SYSTEM FLASH_Lecture (* Remote Flasher Test System Configuration *)
  (* Standard: 61499-1 *)
  (* Version 0.1, 2009-03-05, JHC, Holobloc Inc., Deleted Application. *)
  (* Version 0.0, 2004-01-10, JHC, Rockwell Automation, Modified from FLASHERT_TESTD. *)
  DEVICE CTL_PANEL : FRAME_DEVICE(BOUNDS := [50,100,325,100], GRID := [1,1])
    RESOURCE RES1 : PANEL_RESOURCE
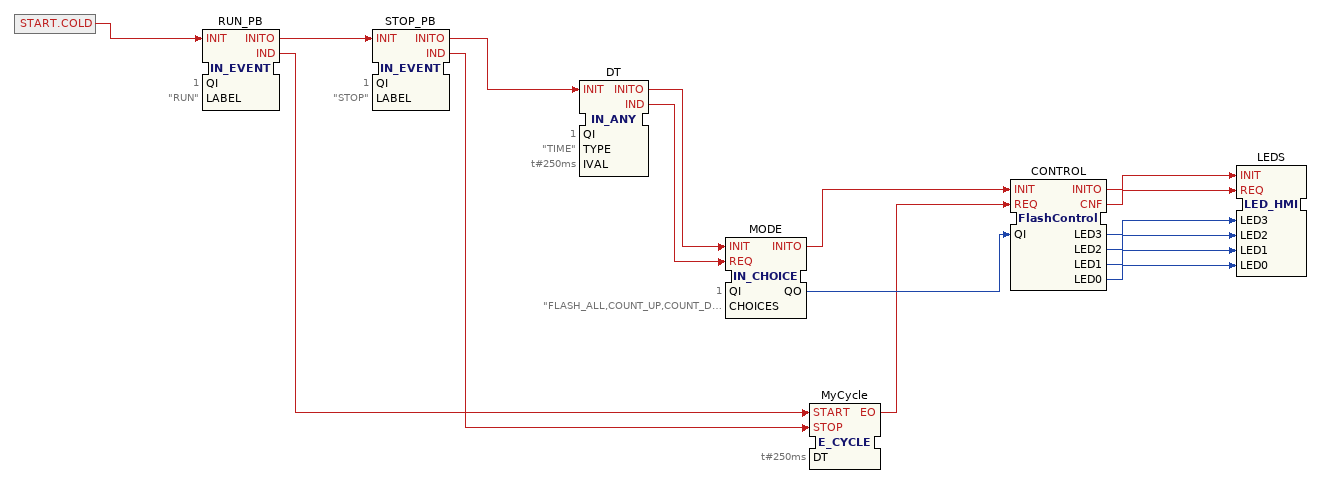
      FBS
        RUN_PB : IN_EVENT(QI := 1, LABEL := "RUN");
        STOP_PB : IN_EVENT(QI := 1, LABEL := "STOP");
        MODE : IN_CHOICE(QI := 1, CHOICES := "FLASH_ALL,COUNT_UP,COUNT_DOWN,CHASE_UP,CHASE_DOWN");
        DT : IN_ANY(QI := 1, TYPE := "TIME", IVAL := t#250ms);
        LEDS : LED_HMI;
        MyCycle : E_CYCLE(DT := t#250ms);
        CONTROL : FlashControl;
      END_FBS
      EVENT_CONNECTIONS
        START.COLD TO RUN_PB.INIT;
        RUN_PB.INITO TO STOP_PB.INIT;
        STOP_PB.INITO TO DT.INIT;
        DT.INITO TO MODE.INIT;
        DT.IND TO MODE.REQ;
        RUN_PB.IND TO MyCycle.START;
        STOP_PB.IND TO MyCycle.STOP;
        MODE.INITO TO CONTROL.INIT;
        CONTROL.INITO TO LEDS.INIT;
        CONTROL.CNF TO LEDS.REQ;
        MyCycle.EO TO CONTROL.REQ;
      END_CONNECTIONS
      DATA_CONNECTIONS
        CONTROL.LED3 TO LEDS.LED3;
        CONTROL.LED2 TO LEDS.LED2;
        CONTROL.LED1 TO LEDS.LED1;
        CONTROL.LED0 TO LEDS.LED0;
        MODE.QO TO CONTROL.QI;
      END_CONNECTIONS
    END_RESOURCE
  END_DEVICE
END_SYSTEM
